{attribute 'GeneratedUsingTerminal: EPP3204-0002-0016'}
{attribute addProperty BoxType "EPP3204-0002-0016"}
{attribute addProperty Id "StatusAT %I*Status_B07533568ValueAT %I*INT2"}
{attribute addProperty CRC "2833212643"}
{attribute addProperty Size "10"}
TYPE RTD_RTDInputs_Channel_A8DF64E3 :
STRUCT
	{attribute addProperty Name "Status"}
	Status AT %I* : Status_B0753356;
	{attribute addProperty Name "Value"}
	Value AT %I* : INT;
END_STRUCT
END_TYPE

(* stored: Version 1.2.0.0, ProductVersion 3.1.4024.9
   DUT RTD_RTDInputs_Channel_A8DF64E3: Id {32b8e4a7-1098-4a2e-852a-6c4da3a6c82f} *)
